PROGRAM PRG_FSV
VAR
	fastFaultSaveMyLife : FB_FastFault;
END_VAR


TV1K4_VFS_1(
	i_xPMPS_OK:= TRUE, 
	i_xExt_OK:= TRUE, 
	i_xVeto:=TRUE,
	i_sDevName:= 'TV1K4:VFS:01', 
	io_fbFFHWO:= g_FastFaultOutput3 );
	

MR3K4_KBO_VFS_1(
	i_xPMPS_OK:= TRUE, 
	i_xExt_OK:= TRUE, 
	i_sDevName:= 'MR3K4:KBO:VFS:1',
	io_fbFFHWO:= g_FastFaultOutput4
);

MR4K4_KBO_VFS_1(
	i_xPMPS_OK:= TRUE, 
	i_xExt_OK:= TRUE, 
	i_sDevName:= 'MR4K4:KBO:VFS:1',
	io_fbFFHWO:= g_FastFaultOutput4
);
(*FastFaultOuput*)	
g_FastFaultOutput3.Execute(bAutoReset:= TRUE);

g_FastFaultOutput4.Execute(i_xVeto:=PMPS_GVL.stCurrentBeamParameters.aStoppers[K_Stopper.ST3K4], bAutoReset:= TRUE);

//g_FastFaultOutput4.q_xFastFaultOut R= NOT g_FastFaultOutput3.q_xFastFaultOut;
//fastFaultSaveMyLife(i_xOK := g_FastFaultOutput3.q_xFastFaultOut, i_xAutoReset := TRUE, io_fbFFHWO:=g_FastFaultOutput4);

//g_FastFaultOutput4.Execute(bAutoReset:= TRUE);

END_PROGRAM

(* stored: Version 1.1.0.1, ProductVersion 3.1.4022.18
   POU PRG_FSV: Id {223741e2-9659-48ba-be92-e06c66eee1cf}, SpecialFunc None *)
